(* IEC 61131-3 sources: Industry-PLC-LLM/data/PLCBEAD_repo/PLCBEAD_PLCEmbed-main/PLC-BEAD/Source/GEB/building_BLIND_CONTROL_S, 1 file *)

(* ---- BLIND_CONTROL_S.ST ---- *)
FUNCTION UDINT_TO_TIME2:TIME

	VAR_INPUT
		IN :	UDINT;
	END_VAR

	UDINT_TO_TIME2 := DINT_TO_TIME(UDINT_TO_DINT(IN));

END_FUNCTION

FUNCTION_BLOCK T_PLC_MS_block
	VAR_OUTPUT
		T_PLC_MS :	UDINT;
	END_VAR

	VAR
		PLC_TICKS_PER_SEC :	INT;
		PLC_SYS_TICK_CNT :	DINT;
	END_VAR

	VAR
		debug :	BOOL;(*Debug-Mode ON / OFF*)
		N :	INT;(*Debug-Faktor*)
		Offset :	UDINT;(*Debug-Offset*)
		temp :	DWORD := DWORD#1;(*Debug-Offset*)
		MODE :	BOOL;(*modus*)
		faktor :	UDINT;(*Systemtakt-Faktor*)
		init :	BOOL;
		v_plc_ticks_per_sec :	UDINT;
		base :	UDINT := UDINT#1000;
	END_VAR

	IF init = FALSE THEN
		v_plc_ticks_per_sec := INT_TO_UDINT(PLC_TICKS_PER_SEC);
		IF v_plc_ticks_per_sec = UDINT#1024 THEN
			faktor := UDINT#1;
			MODE := FALSE;
		ELSIF v_plc_ticks_per_sec > UDINT#0 THEN
			IF v_plc_ticks_per_sec <= base THEN
				faktor := base / v_plc_ticks_per_sec;
				MODE := FALSE;
			ELSE
				faktor := v_plc_ticks_per_sec / base;
				MODE := TRUE;
			END_IF;
		ELSE
			faktor := UDINT#1;
		END_IF;
		init := TRUE;
	END_IF;

	IF MODE THEN
		T_PLC_MS := DINT_TO_UDINT(PLC_SYS_TICK_CNT) / faktor;
	ELSE
		T_PLC_MS := DINT_TO_UDINT(PLC_SYS_TICK_CNT) * faktor;
	END_IF;

	IF debug THEN
		T_PLC_MS := (DWORD_TO_UDINT(SHL(UDINT_TO_DWORD(T_PLC_MS),N) OR SHL(temp,N)) - UDINT#1) + Offset;
	END_IF;
END_FUNCTION_BLOCK

FUNCTION TIME_TO_UDINT2:UDINT
	VAR_INPUT
		X :	TIME;
	END_VAR

	TIME_TO_UDINT2 := DINT_TO_UDINT(TIME_TO_DINT(X));
END_FUNCTION

FUNCTION FRMP_B:BYTE
	VAR_INPUT
		START :	BYTE;
		DIR :	BOOL;
		TD :	TIME;
		TR :	TIME;
	END_VAR

	IF TD < TR THEN
		FRMP_B := MIN(UDINT_TO_BYTE(DWORD_TO_UDINT(SHL(TIME_TO_DWORD(TD), 8)) / TIME_TO_UDINT2(TR)), SEL(DIR, START, USINT_TO_BYTE(USINT#255 - BYTE_TO_USINT(START))));
		IF DIR THEN
			FRMP_B := USINT_TO_BYTE(BYTE_TO_USINT(START) + BYTE_TO_USINT(FRMP_B));
		ELSE
			FRMP_B := USINT_TO_BYTE(BYTE_TO_USINT(START) - BYTE_TO_USINT(FRMP_B));
		END_IF;
	ELSE
		FRMP_B := SEL(DIR, BYTE#0, BYTE#255);
	END_IF;
END_FUNCTION

FUNCTION_BLOCK _RMP_B
	VAR_INPUT
		DIR :	BOOL;
		E :	BOOL := TRUE;
		TR :	TIME;
	END_VAR

	VAR_IN_OUT
		RMP :	BYTE;
	END_VAR

	VAR
		T_PLC_MS :	T_PLC_MS_block;
		TX :	TIME;
		TL :	TIME;
		tn :	TIME;
		init :	BOOL;
		last_DIR :	BOOL;
		START :	BYTE;
	END_VAR

	T_PLC_MS();
	TX := UDINT_TO_TIME(T_PLC_MS.T_PLC_MS);

	IF E AND init AND (DIR = last_DIR) AND (RMP <> SEL(DIR, BYTE#0, BYTE#255)) AND TR = tn THEN
		RMP := FRMP_B(START, DIR, SUB_TIME(TX, TL), TR);
	ELSE
		init := TRUE;
		TL := TX;
		tn := tr;
		START := RMP;
	END_IF;
	last_DIR := DIR;
END_FUNCTION_BLOCK

FUNCTION_BLOCK TREND_DW
	VAR_INPUT
		X :	DWORD;
	END_VAR
	VAR_OUTPUT
		Q :	BOOL;
		TU :	BOOL;
		TD :	BOOL;
		D :	DWORD;
	END_VAR

	VAR
		LAST_X :	DWORD;
	END_VAR

	IF X > last_X THEN
		TU := TRUE;
		TD := FALSE;
		D := UDINT_TO_DWORD(DWORD_TO_UDINT(X) - DWORD_TO_UDINT(last_X));
		Q := TRUE;
	ELSIF X < last_X THEN
		TD := TRUE;
		TU := FALSE;
		D := UDINT_TO_DWORD(DWORD_TO_UDINT(last_X) - DWORD_TO_UDINT(X));
		Q := FALSE;
	ELSE
		TU := FALSE;
		TD := FALSE;
		D := DWORD#0;
	END_IF;
	last_X := X;
END_FUNCTION_BLOCK

FUNCTION_BLOCK _RMP_NEXT
	VAR_INPUT
		E :	BOOL := TRUE;
		IN :	BYTE;
		TR :	TIME;
		TF :	TIME;
		TL :	TIME;
	END_VAR

	VAR_OUTPUT
		DIR :	BOOL;
		UP :	BOOL;
		DN :	BOOL;
	END_VAR

	VAR_IN_OUT
		OUT :	BYTE;
	END_VAR
	VAR
		rmx :	_RMP_B;
		DIRx :	TREND_DW;
		t_lock :	TP;
		xen :	BOOL;
		xDIR :	BOOL;
	END_VAR

	DIRx(X := BYTE_TO_DWORD(IN));

	t_lock(IN := FALSE, PT := TL);

	IF DIRx.TU AND (OUT < IN) THEN
		IF NOT xDIR AND xen THEN t_lock(IN := TRUE); END_IF;
		xen := TRUE;
		xDIR := TRUE;
	ELSIF DIRx.TD AND (OUT > IN) THEN
		IF xDIR AND xen THEN t_lock(IN := TRUE); END_IF;
		xen := TRUE;
		xDIR := FALSE;
	ELSIF xen THEN
		IF (xDIR AND (OUT >= IN)) OR (NOT xDIR AND (OUT <= IN)) THEN
			xen := FALSE;
			IF TL > t#0s THEN t_lock(IN := TRUE); END_IF;
		END_IF;
	END_IF;

	IF NOT t_lock.Q AND xen THEN
		UP := XDIR;
		DIR := XDIR;
		DN := NOT XDIR;
	ELSE
		UP := FALSE;
		DN := FALSE;
	END_IF;

	rmx(rmp := OUT, E := E AND (UP OR DN) , DIR := DIR, tr := SEL(DIR, TF, TR));
	OUT := rmx.RMP;
END_FUNCTION_BLOCK

FUNCTION _BYTE_TO_INT:INT
	VAR_INPUT
		IN :	BYTE;
	END_VAR

	_BYTE_TO_INT := USINT_TO_INT(BYTE_TO_USINT(IN));
END_FUNCTION

FUNCTION_BLOCK BLIND_CONTROL_S_Block

	VAR_INPUT
		UP :	BOOL;
		DN :	BOOL;
		S_IN :	BYTE := BYTE#125;
		PI :	BYTE;
		T_UP :	TIME;
		T_DN :	TIME;
		RU :	BOOL;
		RD :	BOOL;
		T_LOCKOUT :	TIME := T#100ms;
		T_EXT :	TIME;
		EXT_TRIG :	BYTE := BYTE#5;
		R_POS_TOP :	BYTE := BYTE#255;
		R_POS_BOT :	BYTE;
	END_VAR

	VAR_OUTPUT
		POS :	BYTE;
		MU :	BOOL;
		MD :	BOOL;
		STATUS :	BYTE;
	END_VAR

	VAR
		T_PLC_MS :	T_PLC_MS_block;
		rmp :	_RMP_NEXT;
		TX :	TIME;
		last :	TIME;
		pi_last :	BYTE;
	END_VAR

	T_PLC_MS();
	TX:= UDINT_TO_TIME(T_PLC_MS.T_PLC_MS);

	IF UP  AND NOT DN THEN
		rmp.IN := BYTE#255;
		STATUS := BYTE#121;
	ELSIF DN AND NOT UP THEN
		rmp.IN := BYTE#0;
		STATUS := BYTE#122;
	ELSIF NOT (UP OR DN) THEN
		rmp.IN := PI;
		STATUS := S_IN;
	END_IF;

	rmp(E := UP OR DN, TR := T_UP, TF := T_DN, TL := T_LOCKOUT, OUT := POS);
	POS := rmp.OUT;

	CASE _BYTE_TO_INT(STATUS) OF
		0:
			last := TX;
			PI_last := PI XOR BYTE#255;
			STATUS := BYTE#128;

		121:
			MU := TRUE;
			MD := FALSE;
			IF POS >= USINT_TO_BYTE(USINT#255 - BYTE_TO_USINT(EXT_TRIG)) THEN
				POS := BYTE#255;
				last := TX;
				STATUS := BYTE#129;
			END_IF;

		122:
			MD := TRUE;
			MU := FALSE;
			IF POS <= EXT_TRIG THEN
				POS := BYTE#0;
				last := TX;
				STATUS := BYTE#129;
			END_IF;

		123:
			MD := rmp.DN;
			MU := rmp.UP;
			IF NOT (rmp.DN OR rmp.UP) THEN
				IF POS <= EXT_TRIG THEN
					MD := TRUE;
					last := TX;
					STATUS := BYTE#129;
				ELSIF POS >= USINT_TO_BYTE(USINT#255 - BYTE_TO_USINT(EXT_TRIG)) THEN
					MU := TRUE;
					last := TX;
					STATUS := BYTE#129;
				ELSE
					STATUS := S_IN;
				END_IF;
			END_IF;

		124:
			MD := rmp.DN;
			MU := rmp.UP;
			IF NOT(rmp.DN OR rmp.UP) THEN
				PI_last := PI;
				STATUS := S_IN;
			END_IF;

		127:
			IF (SUB_TIME(TX, last)) >= T_LOCKOUT THEN
					STATUS := S_IN;
			END_IF;

		128:
			MU := TRUE;
			MD := FALSE;
			rmp.IN := BYTE#255;
			IF (SUB_TIME(TX, last)) >= (T_UP +  T_EXT) THEN
				MU := FALSE;
				last := TX;
				STATUS := BYTE#127;
			END_IF;

		129:
			IF (SUB_TIME(TX, last)) >= T_EXT THEN
				MU := FALSE;
				MD := FALSE;
				last := TX;
				STATUS := BYTE#127;
			END_IF;

	ELSE
		MU := FALSE;
		MD := FALSE;
		IF PI <> PI_last THEN
			PI_last := PI;
			rmp.IN := PI;
			STATUS := BYTE#123;
		ELSIF POS = BYTE#0 AND RU THEN
			rmp.IN := R_POS_BOT;
			STATUS := BYTE#124;
		ELSIF POS = BYTE#255 AND RD THEN
			rmp.IN := R_POS_TOP;
			STATUS := BYTE#124;
		ELSE
			STATUS := S_IN;
		END_IF;
	END_CASE;

END_FUNCTION_BLOCK

PROGRAM program0
	VAR
		UP :	BOOL;
		DN :	BOOL;
		S_IN :	BYTE := BYTE#125;
		PI :	BYTE;
		T_UP :	TIME;
		T_DN :	TIME;
		RU :	BOOL;
		RD :	BOOL;
		T_LOCKOUT :	TIME := T#100ms;
		T_EXT :	TIME;
		EXT_TRIG :	BYTE := BYTE#5;
		R_POS_TOP :	BYTE := BYTE#255;
		R_POS_BOT :	BYTE;
		POS :	BYTE;
		MU :	BOOL;
		MD :	BOOL;
		STATUS :	BYTE;
		func_block : BLIND_CONTROL_S_Block;
	END_VAR
	func_block.UP := UP;
	func_block.DN := DN;
	func_block.S_IN := S_IN ;
	func_block.PI    := PI    ;
	func_block.T_UP := T_UP;
	func_block.T_DN := T_DN ;
	func_block.RU    := RU    ;
	func_block.RD := RD;
	func_block.T_LOCKOUT := T_LOCKOUT;
	func_block.T_EXT := T_EXT ;
	func_block.EXT_TRIG    := EXT_TRIG    ;
	func_block.R_POS_TOP := R_POS_TOP;
	func_block.R_POS_BOT := R_POS_BOT ;
	func_block();
	POS  := func_block.POS;
	MU  := func_block.MU;
	MD  := func_block.MD;
	STATUS  := func_block.STATUS;
END_PROGRAM
